# EPICS autosave request: iocBoot/iocLTC2983/autosave/pv-spi02-b.req
$(SNAME):CH13:if
